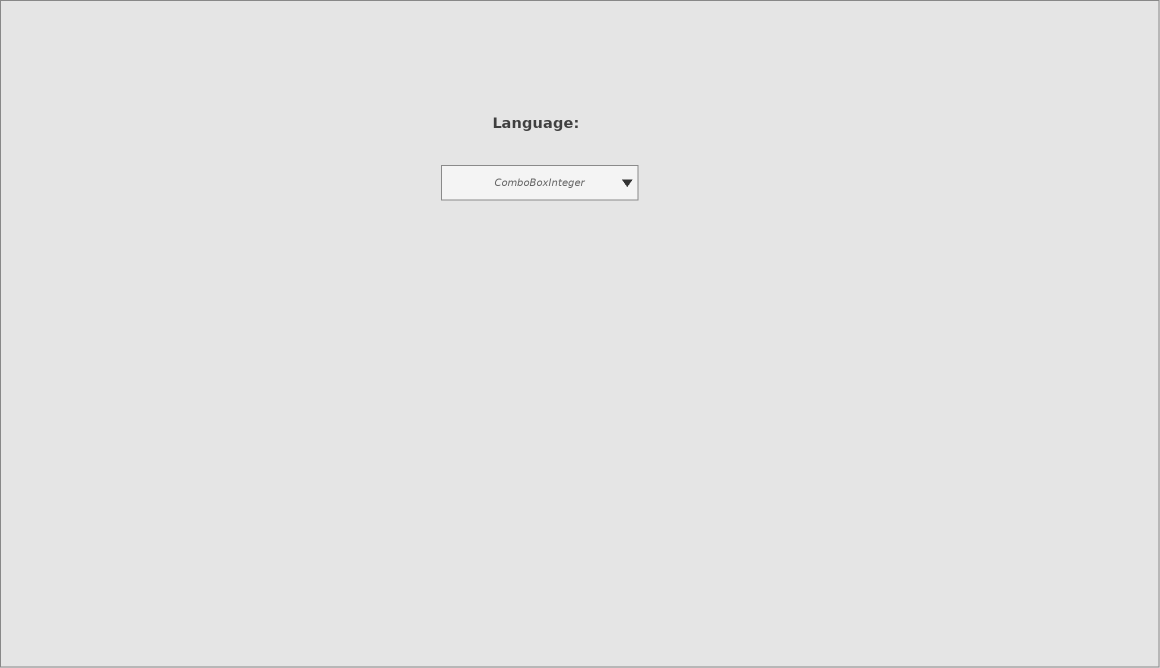
VISUALIZATION V_Settings  // 1160x668
    ComboBoxInteger (441,165 197x35), variable: GVL_HMI.iLang, text list: 'TL_Lang'
    Rectangle (443,100 186x46), "Language:"
END_VISUALIZATION

(* stored: Version 1.1.0.1, ProductVersion 3.1.4024.3
   Visu V_Settings: Id {ba12e61d-bfef-47ad-9c7e-70ffb8fdb4f2} *)
